FUNCTION_BLOCK OUT_ANY_CONSOLE
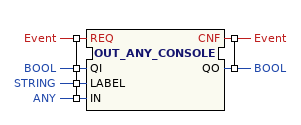
  EVENT_INPUT
    REQ WITH QI, IN, LABEL;
  END_EVENT
  EVENT_OUTPUT
    CNF WITH QO;
  END_EVENT
  VAR_INPUT
    QI : BOOL;
    LABEL : STRING;
    IN : ANY;
  END_VAR
  VAR_OUTPUT
    QO : BOOL;
  END_VAR
END_FUNCTION_BLOCK
